INTERFACE ITF_Base EXTENDS __System.IQueryInterface

PROPERTY Busy : BOOL
GET
END_GET
SET
END_SET
END_PROPERTY

PROPERTY Done : BOOL
GET
END_GET
SET
END_SET
END_PROPERTY

PROPERTY Enable : BOOL
GET
END_GET
SET
END_SET
END_PROPERTY

PROPERTY Error : BOOL
GET
END_GET
SET
END_SET
END_PROPERTY

PROPERTY ErrorID : UINT
GET
END_GET
SET
END_SET
END_PROPERTY

PROPERTY ErrorLevel : E_ErrorLevel
GET
END_GET
SET
END_SET
END_PROPERTY

PROPERTY ErrorMessage : STRING
GET
END_GET
SET
END_SET
END_PROPERTY

PROPERTY ErrorOwner : STRING
GET
END_GET
SET
END_SET
END_PROPERTY

PROPERTY ID : UINT
GET
END_GET
SET
END_SET
END_PROPERTY

METHOD mClearError : BOOL
VAR_INPUT
END_VAR
END_METHOD

METHOD mEnable : bool
VAR_INPUT
END_VAR
END_METHOD

METHOD mError : BOOL
VAR_INPUT
	I_sMessage   : STRING;
	I_eLevel		 : E_ErrorLevel;
	I_uiError		 : UINT;
END_VAR
END_METHOD

METHOD mInit : bool
VAR_INPUT

END_VAR
END_METHOD

METHOD mReset : BOOL
VAR_INPUT
	
END_VAR
END_METHOD

PROPERTY Name : STRING
GET
END_GET
SET
END_SET
END_PROPERTY

END_INTERFACE

(* stored: Version 1.1.0.1, ProductVersion 3.1.4026.18
   Itf ITF_Base: Id {b8e790ab-88dc-4e8a-9453-8571cfddc0b1}
   Folder 01 Properties: Id {8cfcbf18-ccab-4e11-ae93-302bdc03a096}
   Folder 010 Error: Id {a78ccd4f-52d8-4b54-93cc-95ccf21a8219}
   Folder 02 Methods: Id {58c78d7a-3189-4f61-aee0-b0b338a6654b}
   Property Busy: Id {62e63f49-6de4-44af-a604-ded26ddf34bf}
   Get Get: Id {ecb8a7db-351a-42ef-bd50-2252ae379312}
   Set Set: Id {93c5edf2-d26e-4ede-9bbc-78ab60a49e35}
   Property Done: Id {1e4ab53a-0e9a-4d0a-880c-d4463066d983}
   Get Get: Id {af4c7049-93e0-48e1-9787-cbce5805ec32}
   Set Set: Id {a14b88ea-5801-4d28-ac10-a622d186d748}
   Property Enable: Id {bb2da22e-3b0c-4af7-9e42-2da54270641b}
   Get Get: Id {40783ae2-04a7-4f80-886f-f86fad1b429e}
   Set Set: Id {ef395cd3-7810-4e31-9422-3f8c7c29ed01}
   Property Error: Id {2d516bce-bea1-46c9-96ef-f78315234eeb}
   Get Get: Id {19f38900-7939-4895-81ba-19286b8c39d5}
   Set Set: Id {552c0418-cc76-4620-90b9-6fe891ecd85f}
   Property ErrorID: Id {3c885193-8fbd-4b44-bf73-81ba08e80d53}
   Get Get: Id {22a7ef10-921f-4849-8d77-6bb7e75680df}
   Set Set: Id {8b2c7313-b918-4123-b3e0-8236ef720228}
   Property ErrorLevel: Id {851c99a9-8c7a-4bac-94ac-364e10a363b9}
   Get Get: Id {57f75db8-a19f-44b5-8d02-d4fc3b54effb}
   Set Set: Id {d721bb73-c95a-426b-8538-837cdf9656b1}
   Property ErrorMessage: Id {d758939e-80c6-4a4e-844b-488b1154fd70}
   Get Get: Id {d347e905-aa82-458c-88b6-72488f0758cb}
   Set Set: Id {3ebb4141-9cd1-48bc-9fde-14bd36abcde8}
   Property ErrorOwner: Id {c4931aae-b448-42af-9ed8-03c683c13813}
   Get Get: Id {15c60186-dbd6-4f15-80f6-427ab8c56e6b}
   Set Set: Id {f3afcb0c-1942-4135-aa33-4a054b303c51}
   Property ID: Id {ad0a4043-e42e-4d20-9ce4-fe30fc8f1fbe}
   Get Get: Id {1b90543e-090d-4a5d-9a8f-674d12843708}
   Set Set: Id {e8faa49c-6c91-44de-8b58-155f8d8ec86d}
   Method mClearError: Id {0a7eb333-151e-426e-b262-cd2684e19ed8}
   Method mEnable: Id {6edf3d3e-219e-4c99-923f-3d20af9a8e15}
   Method mError: Id {8704c5f7-6efa-476b-b70f-66a367fc6c11}
   Method mInit: Id {bbdaf058-85bc-4ba2-92aa-d7abde21db21}
   Method mReset: Id {67d5ec4b-e405-4638-aa78-3fc040c49139}
   Property Name: Id {aa1dd5da-a811-48f9-a864-c931e827774b}
   Get Get: Id {da106882-2ab2-46b0-b56c-fdb4b6dc941a}
   Set Set: Id {4b510163-e23b-473c-bbff-d41ec26d3f09} *)
